(* Logix 5000 project; controller HP_SSC01 vendor 1 type 14 code 67 rev 17.7; software revision 17.01; part 14 of 15 *)
(* tags used below, declared in another part *)
   A_C2_0200 : ALIAS FOR S_C2_FaultSafety.0;
   A_C2_0201 : ALIAS FOR S_C2_FaultSafety.1;
   A_C2_0202 : ALIAS FOR S_C2_FaultSafety.2;
   A_C2_0203 : ALIAS FOR S_C2_FaultSafety.3;
   A_C2_0204 : ALIAS FOR S_C2_FaultSafety.4;
   A_C2_0206 : ALIAS FOR S_C2_FaultSafety.6;
   A_C2_0208 : ALIAS FOR S_C2_FaultSafety.8;
   A_C2_0209 : ALIAS FOR S_C2_FaultSafety.9;
   A_C2_0210 : ALIAS FOR S_C2_FaultSafety.10;
   A_C2_0211 : ALIAS FOR S_C2_FaultSafety.11;
   A_C2_0216 : ALIAS FOR S_C2_FaultSafety.16;
   A_C2_0217 : ALIAS FOR S_C2_FaultSafety.17;
   A_C2_0220 : ALIAS FOR S_C2_FaultSafety.20;
   A_C3_0200 : ALIAS FOR S_C3_FaultSafety.0;
   A_C3_0201 : ALIAS FOR S_C3_FaultSafety.1;
   A_C3_0202 : ALIAS FOR S_C3_FaultSafety.2;
   A_C3_0203 : ALIAS FOR S_C3_FaultSafety.3;
   A_C3_0204 : ALIAS FOR S_C3_FaultSafety.4;
   A_C3_0206 : ALIAS FOR S_C3_FaultSafety.6;
   A_C3_0208 : ALIAS FOR S_C3_FaultSafety.8;
   A_C3_0209 : ALIAS FOR S_C3_FaultSafety.9;
   A_C3_0210 : ALIAS FOR S_C3_FaultSafety.10;
   A_C3_0211 : ALIAS FOR S_C3_FaultSafety.11;
   A_C3_0216 : ALIAS FOR S_C3_FaultSafety.16;
   A_C3_0217 : ALIAS FOR S_C3_FaultSafety.17;
   A_C3_0218 : ALIAS FOR S_C3_FaultSafety.18;
   A_C3_0219 : ALIAS FOR S_C3_FaultSafety.19;
   A_C3_0220 : ALIAS FOR S_C3_FaultSafety.20;
   A_C3_0221 : ALIAS FOR S_C3_FaultSafety.21;
   A_C3_0222 : ALIAS FOR S_C3_FaultSafety.22;
   A_C3_0223 : ALIAS FOR S_C3_FaultSafety.23;
   A_C3_0224 : ALIAS FOR S_C3_FaultSafety.24;
   A_C3_0230 : ALIAS FOR S_C3_FaultSafety.30;
   A_C3_0231 : ALIAS FOR S_C3_FaultSafety.31;
   A_S01_0104 : ALIAS FOR System_FaultSafeIO.4;
   A_S01_0122 : ALIAS FOR System_FaultSafeIO.22;
   C03_SafeMemory : Udt_Carsl_SafeData;
   C2_EvacInPositionTest : DINT;
   Multiplier : DINT;
   none : BOOL;
   RCS_CMD_EvacToStation : BOOL;
   RCS_SafeMemory_S01 : Udt_RCS_SafeData;
   RCS_SyncMotionEnable : BOOL;
   S1_C3_SafeOffFdbkRIN : REDUNDANT_INPUT;
   S_C1_ModeRemote : BOOL;
   S_C2_AtEvacSpeed : BOOL;
   S_C2_BrakeTest : BOOL;
   S_C2_CircuitReset : BOOL;
   S_C2_CircuitReset_Pulse : TIMER;
   S_C2_DrawBridge_LS1 : ALIAS FOR SSC01_Safe2:I.Pt02Data;
   S_C2_DrawBridge_LS2 : ALIAS FOR SSC01_Safe2:I.Pt03Data;
   S_C2_DrawbridgeInputOK : BOOL;
   S_C2_DrawbridgeRIN : REDUNDANT_INPUT;
   S_C2_DumpTest : BOOL;
   S_C2_EvacOK : BOOL;
   S_C2_ExecuteInputOK : BOOL;
   S_C2_ExecutePB : BOOL;
   S_C2_FaultReset : BOOL;
   S_C2_FaultSafety : DINT;
   S_C2_FaultSafety_OK : BOOL;
   S_C2_FaultStandard : DINT;
   S_C2_FaultStandard_OK : BOOL;
   S_C2_FW_LocalOK : BOOL;
   S_C2_InEvacPosition : BOOL;
   S_C2_MaintEnable : BOOL;
   S_C2_MCC2_LIM_MCR : ALIAS FOR C2_Safe:O.Pt04Data;
   S_C2_ModeLocal : BOOL;
   S_C2_ModeRemote : BOOL;
   S_C2_MotionEnabled : BOOL;
   S_C2_MOTN_EXEC_RIN : REDUNDANT_INPUT;
   S_C2_MOTN_EXEC_SS_A : ALIAS FOR C2_Safe:I.Pt02Data;
   S_C2_MOTN_EXEC_SS_B : ALIAS FOR C2_Safe:I.Pt03Data;
   S_C2_MotorActualPositionX1000 : DINT;
   S_C2_MotorAverageVelocityX1000 : DINT;
   S_C2_MStop : EMERGENCY_STOP;
   S_C2_MSTOP_A : ALIAS FOR C2_Safe:I.Pt06Data;
   S_C2_MSTOP_B : ALIAS FOR C2_Safe:I.Pt07Data;
   S_C2_MSTOP_InputOK : BOOL;
   S_C2_MSTOP_LT : ALIAS FOR C2_Safe:O.Pt02Data;
   S_C2_OIT_FaultReset : BOOL;
   S_C2_ONS : DINT;
   S_C2_ONS_CircuitFault : BOOL;
   S_C2_ONS_Status : BOOL;
   S_C2_OutputEnable : BOOL;
   S_C2_PressureOK : ALIAS FOR C2_Safe:I.Pt05Data;
   S_C2_ResetTOF : TIMER;
   S_C2_SAFE_FDBK_Aux1 : BOOL;
   S_C2_SAFE_FDBK_Aux2 : BOOL;
   S_C2_SAFE_OFF_FDBK1 : ALIAS FOR C2_Safe:I.Pt01Data;
   S_C2_SAFE_OFF_FDBK2 : ALIAS FOR C2_Safe:I.Pt00Data;
   S_C2_SafeOff_ROUT : REDUNDANT_OUTPUT;
   S_C2_SafeOffEnabled : BOOL;
   S_C2_SafeOffEngaged : BOOL;
   S_C2_SafeOffFdbkRIN : REDUNDANT_INPUT;
   S_C2_SafeOffInputOK : BOOL;
   S_C2_SAFETY_ENABLE_1 : ALIAS FOR C2_Safe:O.Pt00Data;
   S_C2_SAFETY_ENABLE_2 : ALIAS FOR C2_Safe:O.Pt01Data;
   S_C2_SS_RemoteMode : BOOL;
   S_C2_Stop0_OK : BOOL;
   S_C2_Stop1_OK : BOOL;
   S_C2_Stop1_OK_TOF : TIMER;
   S_C3_AtEvacSpeed : BOOL;
   S_C3_BrakeRelease : ALIAS FOR C3_Safe:O.Pt06Data;
   S_C3_BrakeReleaseSelected : BOOL;
   S_C3_BrakeTest : BOOL;
   S_C3_CircuitReset : BOOL;
   S_C3_CircuitReset_Pulse : TIMER;
   S_C3_DrawBridge_LS1 : ALIAS FOR SSC01_Safe2:I.Pt06Data;
   S_C3_DrawBridge_LS2 : ALIAS FOR SSC01_Safe2:I.Pt07Data;
   S_C3_DrawbridgeInputOK : BOOL;
   S_C3_DrawbridgeRIN : REDUNDANT_INPUT;
   S_C3_DumpValveRelease : ALIAS FOR C3_Safe:O.Pt05Data;
   S_C3_DumpValveReleaseSelected : BOOL;
   S_C3_EncoderBuffer : DINT[4];
   S_C3_EncoderChange : DINT;
   S_C3_EncoderCounter : DINT;
   S_C3_EncoderCounts : DINT;
   S_C3_EncoderDegree : DINT;
   S_C3_EncoderPositionAtHome : DINT;
   S_C3_EncoderPositionAtHomeSet : BOOL;
   S_C3_EncoderRev : DINT;
   S_C3_EncoderRevX1000 : DINT;
   S_C3_EncoderTemp : DINT;
   S_C3_EncoderTemp2 : DINT;
   S_C3_EvacOK : BOOL;
   S_C3_ExecuteInputOK : BOOL;
   S_C3_ExecutePB : BOOL;
   S_C3_FaultReset : BOOL;
   S_C3_FaultSafety : DINT;
   S_C3_FaultSafety_OK : BOOL;
   S_C3_FaultStandard_OK : BOOL;
   S_C3_FaultTimer : TIMER[8];
   S_C3_Homed : BOOL;
   S_C3_HomeInputStatus : BOOL;
   S_C3_HomeSafePE : ALIAS FOR C3_Safe:I.Pt04Data;
   S_C3_InEvacPosition : BOOL;
   S_C3_ModeLocal : BOOL;
   S_C3_ModeRemote : BOOL;
   S_C3_MOTN_EXEC_RIN : REDUNDANT_INPUT;
   S_C3_MOTN_EXEC_SS_A : ALIAS FOR C3_Safe:I.Pt02Data;
   S_C3_MOTN_EXEC_SS_B : ALIAS FOR C3_Safe:I.Pt03Data;
   S_C3_MotorActualPositionX1000 : DINT;
   S_C3_MotorActualPositionX1000MOD60 : DINT;
   S_C3_MotorAverageVelocityX1000 : DINT;
   S_C3_MotorToEncoderError : DINT;
   S_C3_MStop : EMERGENCY_STOP;
   S_C3_MSTOP_A : ALIAS FOR C3_Safe:I.Pt06Data;
   S_C3_MSTOP_B : ALIAS FOR C3_Safe:I.Pt07Data;
   S_C3_MSTOP_InputOK : BOOL;
   S_C3_NearOnPath : BOOL;
   S_C3_NearOnPathHi : DINT;
   S_C3_NearOnPathHiBase : DINT;
   S_C3_NearOnPathLow : DINT;
   S_C3_NearOnPathLowBase : DINT;
   S_C3_OffPath : BOOL;
   S_C3_OnPath : BOOL;
   S_C3_OnPathHi : DINT;
   S_C3_OnPathLow : DINT;
   S_C3_ONS_CircuitFault : BOOL;
   S_C3_ONS_Fault : BOOL;
   S_C3_OutputEnable : BOOL;
   S_C3_PathError : DINT;
   S_C3_PathErrorTest : DINT;
   S_C3_PathErrorTestTemp : DINT;
   S_C3_PathErrorTestTemp2 : DINT;
   S_C3_PathOffset : DINT;
   S_C3_PressureOK : ALIAS FOR C3_Safe:I.Pt05Data;
   S_C3_RemoteBrakeAndHomeSequence : DINT;
   S_C3_ReverseMotionDebounce : TIMER;
   S_C3_SAFE_FDBK_Aux1 : BOOL;
   S_C3_SAFE_FDBK_Aux2 : BOOL;
   S_C3_SAFE_OFF_FDBK1 : ALIAS FOR C3_Safe:I.Pt01Data;
   S_C3_SAFE_OFF_FDBK2 : ALIAS FOR C3_Safe:I.Pt00Data;
   S_C3_SafeOff_ROUT : REDUNDANT_OUTPUT;
   S_C3_SafeOffEnabled : BOOL;
   S_C3_SafeOffEngaged : BOOL;
   S_C3_SafeOffInputOK : BOOL;
   S_C3_SetEncoderHomePosition : BOOL;
   S_C3_WindowAdderTemp1 : DINT;
   S_C3_WindowAdderTemp2 : DINT;
   S_C3_WindowAdderTemp3 : DINT;
   S_EncoderRollover : DINT;
   S_EvacToStationTON : TIMER;
   S_FlashOn : TIMER;
   S_RCS_CMD_FaultReset : BOOL;
   S_RCS_EvacSpeedStart_TON : TIMER;
   S_RCS_MasterPositionDegrees : DINT;
   S_RCS_MotionEnable : BOOL;
   S_System_FaultStandard : DINT;
   SSC_Rail_BypassOK : BOOL;
   SSC_SafeFlt_OK : BOOL;
   SSC_SafetyIO_OK : BOOL;
   SSC_StdFlt_OK : BOOL;
   SSC_Stop0_OK : BOOL;
   SSC_Stop1_OK : BOOL;
(* SafeCarousel2, continued *)

ROUTINE SC230_SafetyInputs   (* ladder *)
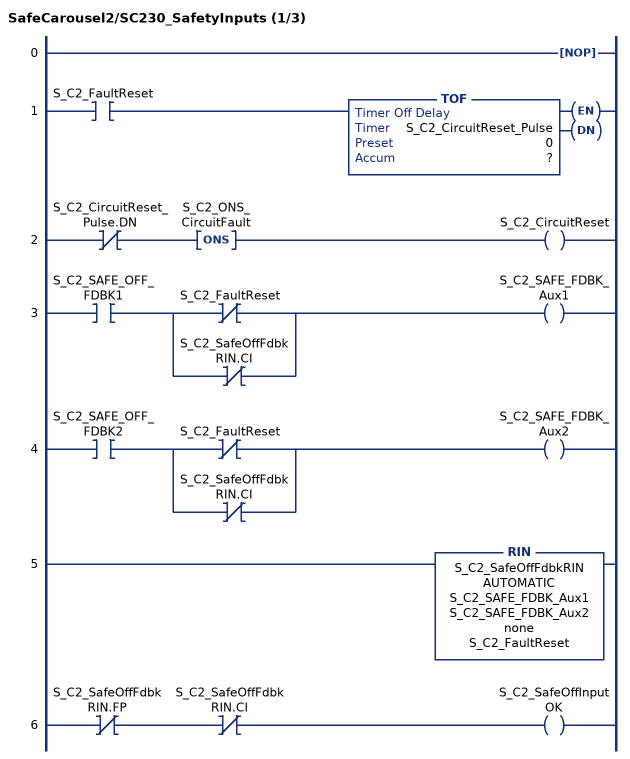
   0: NOP();
   1: XIC(S_C2_FaultReset)TOF(S_C2_CircuitReset_Pulse,?,?);
   2: XIO(S_C2_CircuitReset_Pulse.DN)ONS(S_C2_ONS_CircuitFault)OTE(S_C2_CircuitReset);
   3: XIC(S_C2_SAFE_OFF_FDBK1)[XIO(S_C2_FaultReset) ,XIO(S_C2_SafeOffFdbkRIN.CI) ]OTE(S_C2_SAFE_FDBK_Aux1);
   4: XIC(S_C2_SAFE_OFF_FDBK2)[XIO(S_C2_FaultReset) ,XIO(S_C2_SafeOffFdbkRIN.CI) ]OTE(S_C2_SAFE_FDBK_Aux2);
   5: RIN(S_C2_SafeOffFdbkRIN,AUTOMATIC,S_C2_SAFE_FDBK_Aux1,S_C2_SAFE_FDBK_Aux2,none,S_C2_FaultReset);
   6: XIO(S_C2_SafeOffFdbkRIN.FP)XIO(S_C2_SafeOffFdbkRIN.CI)OTE(S_C2_SafeOffInputOK);
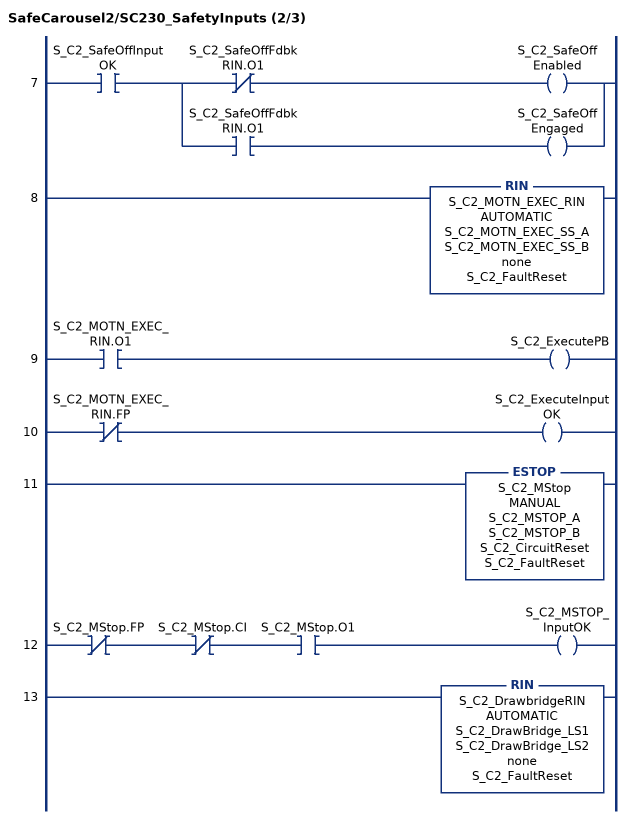
   7: XIC(S_C2_SafeOffInputOK)[XIO(S_C2_SafeOffFdbkRIN.O1) OTE(S_C2_SafeOffEnabled) ,XIC(S_C2_SafeOffFdbkRIN.O1) OTE(S_C2_SafeOffEngaged) ];
   8: RIN(S_C2_MOTN_EXEC_RIN,AUTOMATIC,S_C2_MOTN_EXEC_SS_A,S_C2_MOTN_EXEC_SS_B,none,S_C2_FaultReset);
   9: XIC(S_C2_MOTN_EXEC_RIN.O1)OTE(S_C2_ExecutePB);
   10: XIO(S_C2_MOTN_EXEC_RIN.FP)OTE(S_C2_ExecuteInputOK);
   11: ESTOP(S_C2_MStop,MANUAL,S_C2_MSTOP_A,S_C2_MSTOP_B,S_C2_CircuitReset,S_C2_FaultReset);
   12: XIO(S_C2_MStop.FP)XIO(S_C2_MStop.CI)XIC(S_C2_MStop.O1)OTE(S_C2_MSTOP_InputOK);
   13: RIN(S_C2_DrawbridgeRIN,AUTOMATIC,S_C2_DrawBridge_LS1,S_C2_DrawBridge_LS2,none,S_C2_FaultReset);
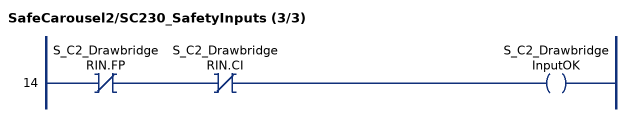
   14: XIO(S_C2_DrawbridgeRIN.FP)XIO(S_C2_DrawbridgeRIN.CI)OTE(S_C2_DrawbridgeInputOK);
END_ROUTINE

ROUTINE SC235_SafetyOutputs   (* ladder *)
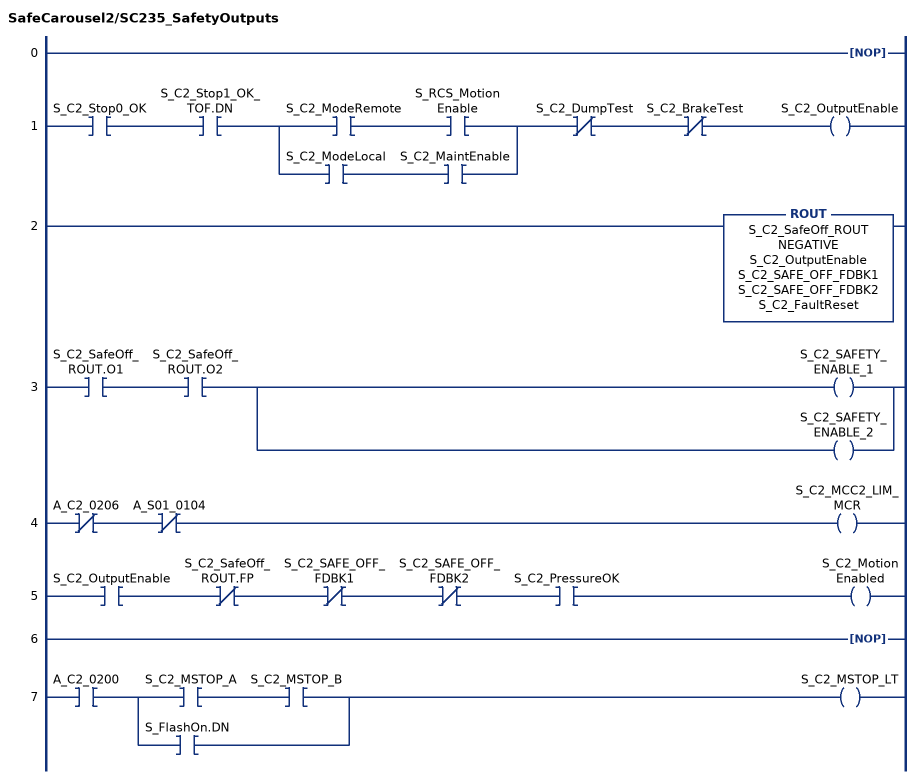
   0: NOP();
   1: XIC(S_C2_Stop0_OK)XIC(S_C2_Stop1_OK_TOF.DN)[XIC(S_C2_ModeRemote) XIC(S_RCS_MotionEnable) ,XIC(S_C2_ModeLocal) XIC(S_C2_MaintEnable) ]XIO(S_C2_DumpTest)XIO(S_C2_BrakeTest)OTE(S_C2_OutputEnable);
   2: ROUT(S_C2_SafeOff_ROUT,NEGATIVE,S_C2_OutputEnable,S_C2_SAFE_OFF_FDBK1,S_C2_SAFE_OFF_FDBK2,S_C2_FaultReset);
   3: XIC(S_C2_SafeOff_ROUT.O1)XIC(S_C2_SafeOff_ROUT.O2)[OTE(S_C2_SAFETY_ENABLE_1) ,OTE(S_C2_SAFETY_ENABLE_2) ];
   4: XIO(A_C2_0206)XIO(A_S01_0104)OTE(S_C2_MCC2_LIM_MCR);
   5: XIC(S_C2_OutputEnable)XIO(S_C2_SafeOff_ROUT.FP)XIO(S_C2_SAFE_OFF_FDBK1)XIO(S_C2_SAFE_OFF_FDBK2)XIC(S_C2_PressureOK)OTE(S_C2_MotionEnabled);
   6: NOP();
   7: XIC(A_C2_0200)[XIC(S_C2_MSTOP_A) XIC(S_C2_MSTOP_B) ,XIC(S_FlashOn.DN) ]OTE(S_C2_MSTOP_LT);
END_ROUTINE

ROUTINE SC240_Status   (* ladder *)
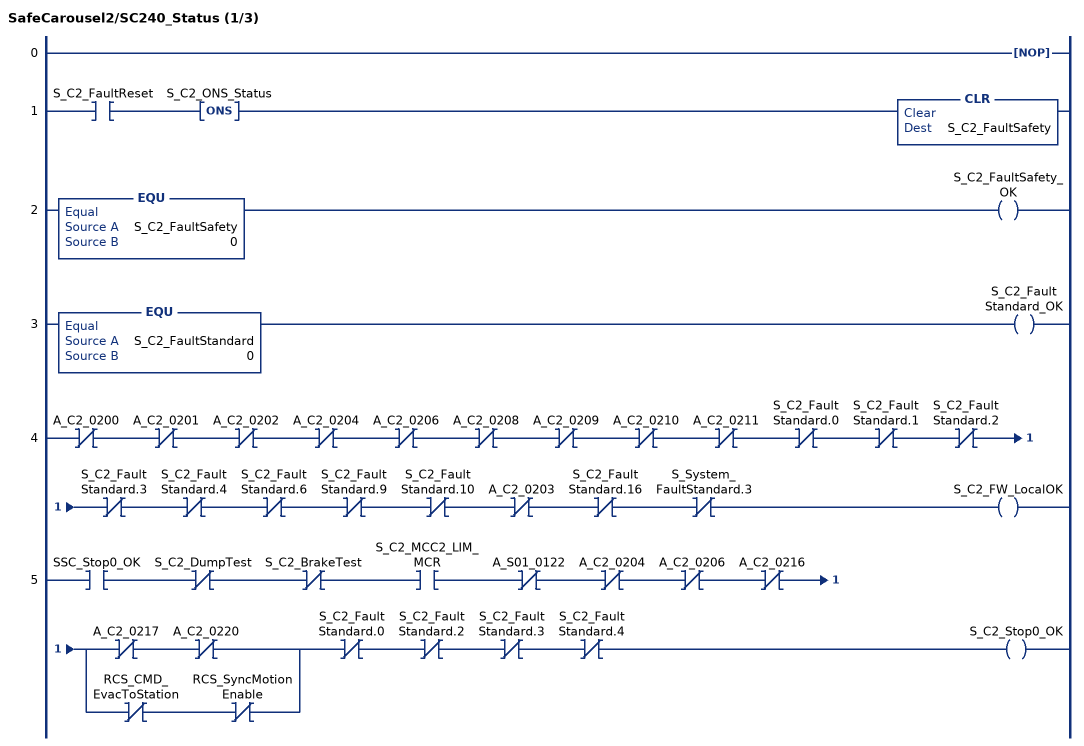
   0: NOP();
   1: XIC(S_C2_FaultReset)ONS(S_C2_ONS_Status)CLR(S_C2_FaultSafety);
   2: EQU(S_C2_FaultSafety,0)OTE(S_C2_FaultSafety_OK);
   3: EQU(S_C2_FaultStandard,0)OTE(S_C2_FaultStandard_OK);
   4: XIO(A_C2_0200)XIO(A_C2_0201)XIO(A_C2_0202)XIO(A_C2_0204)XIO(A_C2_0206)XIO(A_C2_0208)XIO(A_C2_0209)XIO(A_C2_0210)XIO(A_C2_0211)XIO(S_C2_FaultStandard.0)XIO(S_C2_FaultStandard.1)XIO(S_C2_FaultStandard.2)XIO(S_C2_FaultStandard.3)XIO(S_C2_FaultStandard.4)XIO(S_C2_FaultStandard.6)XIO(S_C2_FaultStandard.9)XIO(S_C2_FaultStandard.10)XIO(A_C2_0203)XIO(S_C2_FaultStandard.16)XIO(S_System_FaultStandard.3)OTE(S_C2_FW_LocalOK);
   5: XIC(SSC_Stop0_OK)XIO(S_C2_DumpTest)XIO(S_C2_BrakeTest)XIC(S_C2_MCC2_LIM_MCR)XIO(A_S01_0122)XIO(A_C2_0204)XIO(A_C2_0206)XIO(A_C2_0216)[XIO(A_C2_0217) XIO(A_C2_0220) ,XIO(RCS_CMD_EvacToStation) XIO(RCS_SyncMotionEnable) ]XIO(S_C2_FaultStandard.0)XIO(S_C2_FaultStandard.2)XIO(S_C2_FaultStandard.3)XIO(S_C2_FaultStandard.4)OTE(S_C2_Stop0_OK);
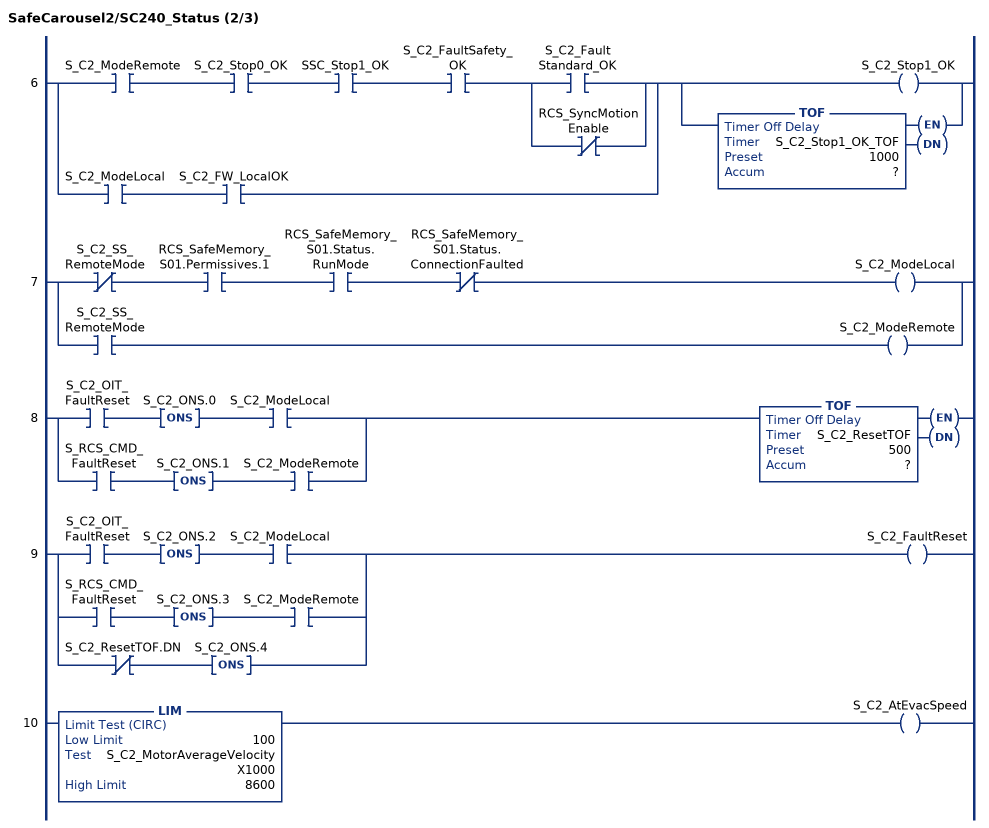
   6: [XIC(S_C2_ModeRemote) XIC(S_C2_Stop0_OK) XIC(SSC_Stop1_OK) XIC(S_C2_FaultSafety_OK) [XIC(S_C2_FaultStandard_OK) ,XIO(RCS_SyncMotionEnable) ] ,XIC(S_C2_ModeLocal) XIC(S_C2_FW_LocalOK) ][OTE(S_C2_Stop1_OK) ,TOF(S_C2_Stop1_OK_TOF,?,?) ];
   7: [XIO(S_C2_SS_RemoteMode) XIC(RCS_SafeMemory_S01.Permissives.1) XIC(RCS_SafeMemory_S01.Status.RunMode) XIO(RCS_SafeMemory_S01.Status.ConnectionFaulted) OTE(S_C2_ModeLocal) ,XIC(S_C2_SS_RemoteMode) OTE(S_C2_ModeRemote) ];
   8: [XIC(S_C2_OIT_FaultReset) ONS(S_C2_ONS.0) XIC(S_C2_ModeLocal) ,XIC(S_RCS_CMD_FaultReset) ONS(S_C2_ONS.1) XIC(S_C2_ModeRemote) ]TOF(S_C2_ResetTOF,?,?);
   9: [XIC(S_C2_OIT_FaultReset) ONS(S_C2_ONS.2) XIC(S_C2_ModeLocal) ,XIC(S_RCS_CMD_FaultReset) ONS(S_C2_ONS.3) XIC(S_C2_ModeRemote) ,XIO(S_C2_ResetTOF.DN) ONS(S_C2_ONS.4) ]OTE(S_C2_FaultReset);
   10: LIM(100,S_C2_MotorAverageVelocityX1000,8600)OTE(S_C2_AtEvacSpeed);
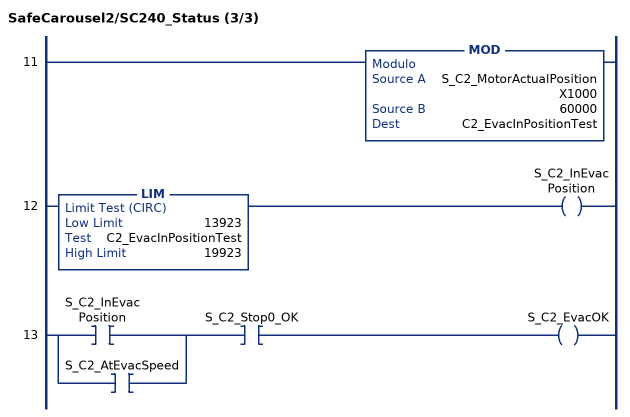
   11: MOD(S_C2_MotorActualPositionX1000,60000,C2_EvacInPositionTest);
   12: LIM(13923,C2_EvacInPositionTest,19923)OTE(S_C2_InEvacPosition);
   13: [XIC(S_C2_InEvacPosition) ,XIC(S_C2_AtEvacSpeed) ]XIC(S_C2_Stop0_OK)OTE(S_C2_EvacOK);
END_ROUTINE
END_PROGRAM

PROGRAM SafeCarousel3   (* main routine SC300_Main *)

ROUTINE SC300_Main   (* ladder *)
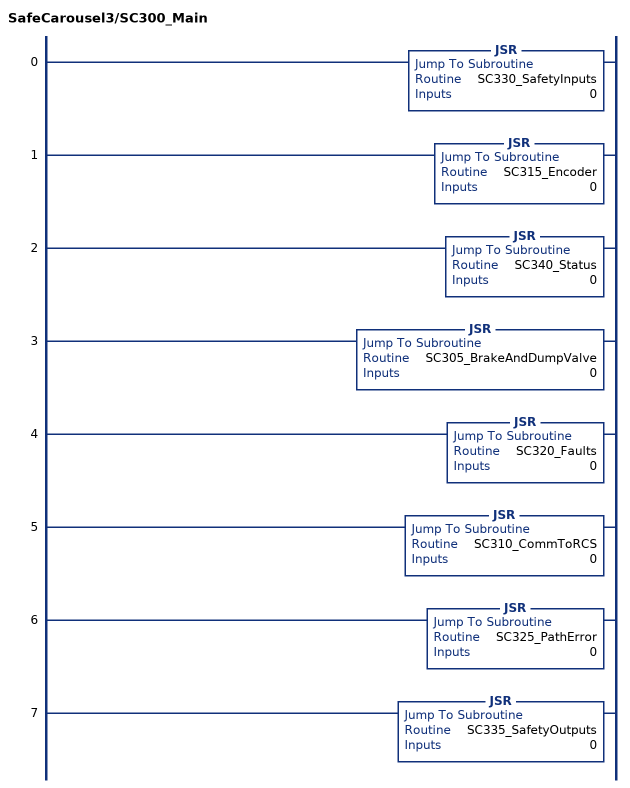
   0: JSR(SC330_SafetyInputs,0);
   1: JSR(SC315_Encoder,0);
   2: JSR(SC340_Status,0);
   3: JSR(SC305_BrakeAndDumpValve,0);
   4: JSR(SC320_Faults,0);
   5: JSR(SC310_CommToRCS,0);
   6: JSR(SC325_PathError,0);
   7: JSR(SC335_SafetyOutputs,0);
END_ROUTINE

ROUTINE SC305_BrakeAndDumpValve   (* ladder *)
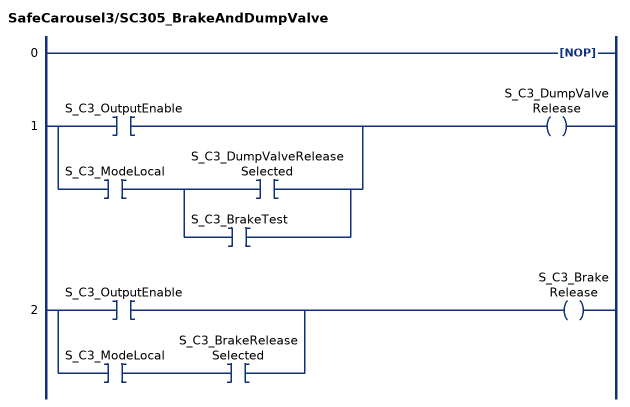
   0: NOP();
   1: [XIC(S_C3_OutputEnable) ,XIC(S_C3_ModeLocal) [XIC(S_C3_DumpValveReleaseSelected) ,XIC(S_C3_BrakeTest) ] ]OTE(S_C3_DumpValveRelease);
   2: [XIC(S_C3_OutputEnable) ,XIC(S_C3_ModeLocal) XIC(S_C3_BrakeReleaseSelected) ]OTE(S_C3_BrakeRelease);
END_ROUTINE

ROUTINE SC310_CommToRCS   (* ladder *)
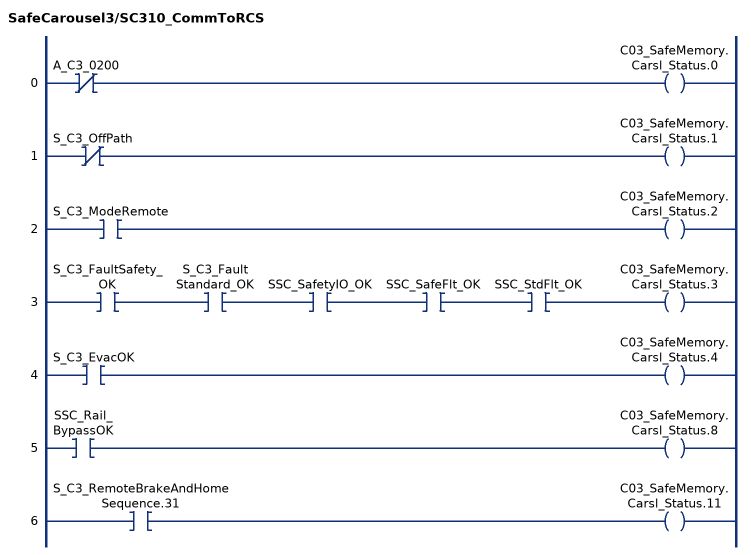
   0: XIO(A_C3_0200)OTE(C03_SafeMemory.Carsl_Status.0);
   1: XIO(S_C3_OffPath)OTE(C03_SafeMemory.Carsl_Status.1);
   2: XIC(S_C3_ModeRemote)OTE(C03_SafeMemory.Carsl_Status.2);
   3: XIC(S_C3_FaultSafety_OK)XIC(S_C3_FaultStandard_OK)XIC(SSC_SafetyIO_OK)XIC(SSC_SafeFlt_OK)XIC(SSC_StdFlt_OK)OTE(C03_SafeMemory.Carsl_Status.3);
   4: XIC(S_C3_EvacOK)OTE(C03_SafeMemory.Carsl_Status.4);
   5: XIC(SSC_Rail_BypassOK)OTE(C03_SafeMemory.Carsl_Status.8);
   6: XIC(S_C3_RemoteBrakeAndHomeSequence.31)OTE(C03_SafeMemory.Carsl_Status.11);
END_ROUTINE

ROUTINE SC315_Encoder   (* ladder *)
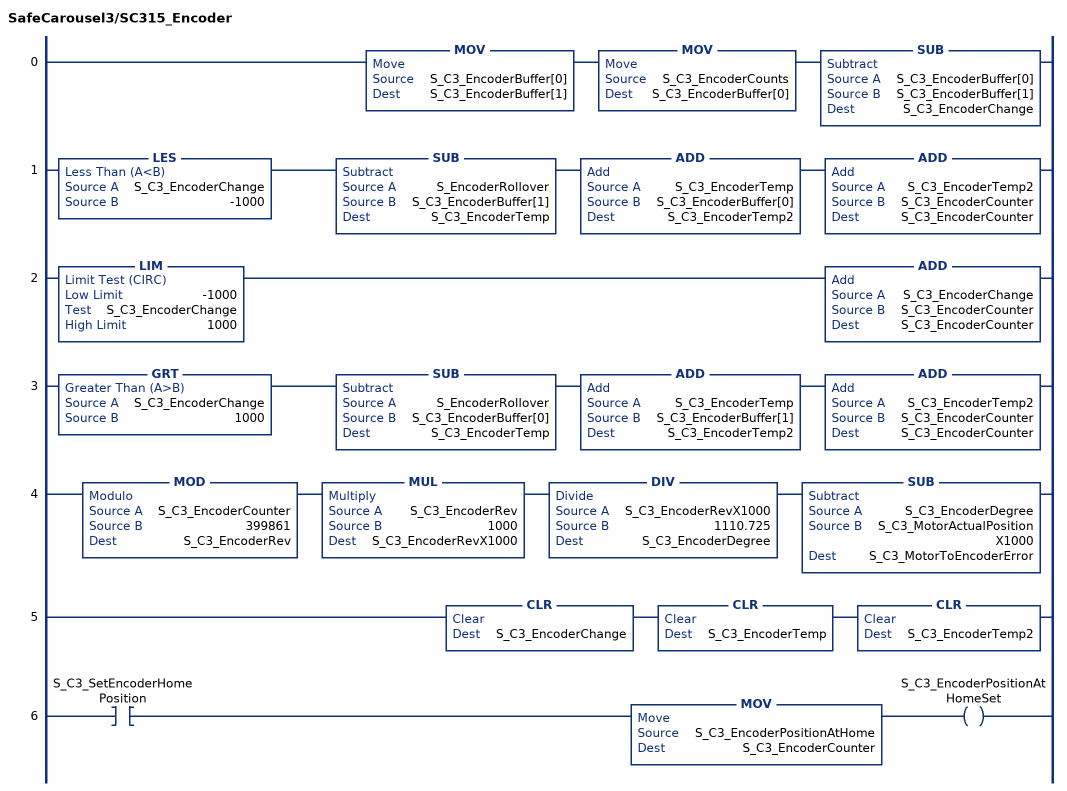
   0: MOV(S_C3_EncoderBuffer[0],S_C3_EncoderBuffer[1])MOV(S_C3_EncoderCounts,S_C3_EncoderBuffer[0])SUB(S_C3_EncoderBuffer[0],S_C3_EncoderBuffer[1],S_C3_EncoderChange);
   1: LES(S_C3_EncoderChange,-1000)SUB(S_EncoderRollover,S_C3_EncoderBuffer[1],S_C3_EncoderTemp)ADD(S_C3_EncoderTemp,S_C3_EncoderBuffer[0],S_C3_EncoderTemp2)ADD(S_C3_EncoderTemp2,S_C3_EncoderCounter,S_C3_EncoderCounter);
   2: LIM(-1000,S_C3_EncoderChange,1000)ADD(S_C3_EncoderChange,S_C3_EncoderCounter,S_C3_EncoderCounter);
   3: GRT(S_C3_EncoderChange,1000)SUB(S_EncoderRollover,S_C3_EncoderBuffer[0],S_C3_EncoderTemp)ADD(S_C3_EncoderTemp,S_C3_EncoderBuffer[1],S_C3_EncoderTemp2)ADD(S_C3_EncoderTemp2,S_C3_EncoderCounter,S_C3_EncoderCounter);
   4: MOD(S_C3_EncoderCounter,399861,S_C3_EncoderRev)MUL(S_C3_EncoderRev,1000,S_C3_EncoderRevX1000)DIV(S_C3_EncoderRevX1000,1110.725,S_C3_EncoderDegree)SUB(S_C3_EncoderDegree,S_C3_MotorActualPositionX1000,S_C3_MotorToEncoderError);
   5: CLR(S_C3_EncoderChange)CLR(S_C3_EncoderTemp)CLR(S_C3_EncoderTemp2);
   6: XIC(S_C3_SetEncoderHomePosition)MOV(S_C3_EncoderPositionAtHome,S_C3_EncoderCounter)OTE(S_C3_EncoderPositionAtHomeSet);
END_ROUTINE

ROUTINE SC320_Faults   (* ladder *)
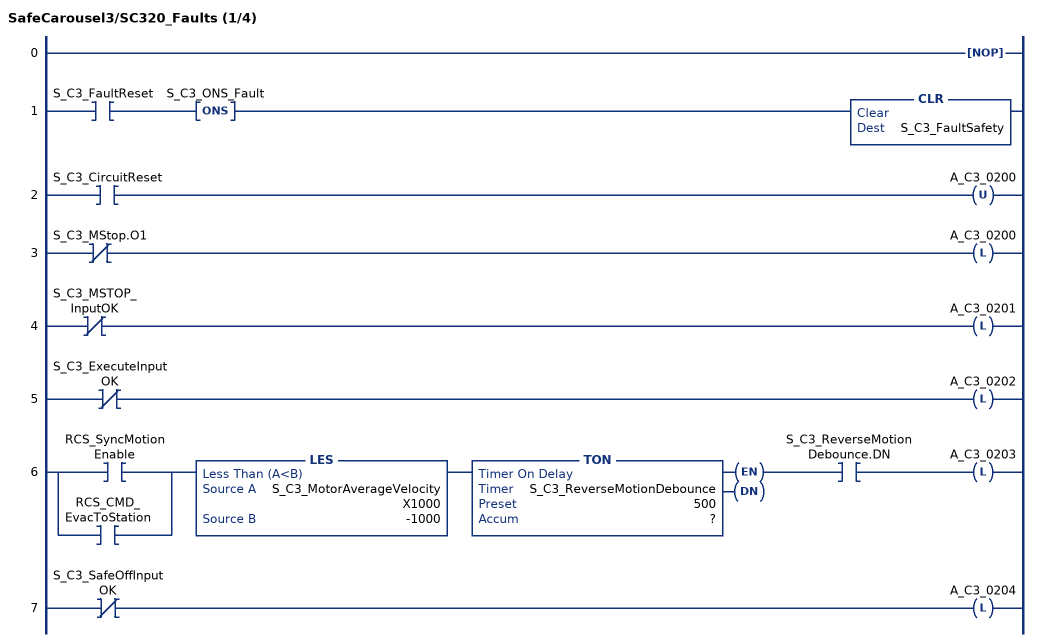
   0: NOP();
   1: XIC(S_C3_FaultReset)ONS(S_C3_ONS_Fault)CLR(S_C3_FaultSafety);
   2: XIC(S_C3_CircuitReset)OTU(A_C3_0200);
   3: XIO(S_C3_MStop.O1)OTL(A_C3_0200);
   4: XIO(S_C3_MSTOP_InputOK)OTL(A_C3_0201);
   5: XIO(S_C3_ExecuteInputOK)OTL(A_C3_0202);
   6: [XIC(RCS_SyncMotionEnable) ,XIC(RCS_CMD_EvacToStation) ]LES(S_C3_MotorAverageVelocityX1000,-1000)TON(S_C3_ReverseMotionDebounce,?,?)XIC(S_C3_ReverseMotionDebounce.DN)OTL(A_C3_0203);
   7: XIO(S_C3_SafeOffInputOK)OTL(A_C3_0204);
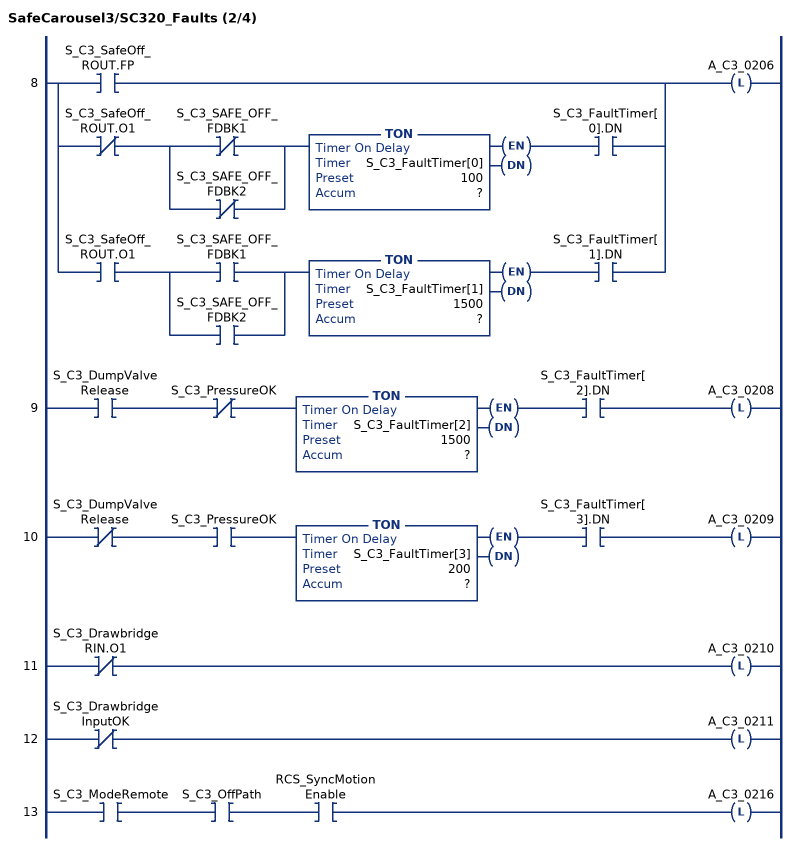
   8: [XIC(S_C3_SafeOff_ROUT.FP) ,XIO(S_C3_SafeOff_ROUT.O1) [XIO(S_C3_SAFE_OFF_FDBK1) ,XIO(S_C3_SAFE_OFF_FDBK2) ] TON(S_C3_FaultTimer[0],?,?) XIC(S_C3_FaultTimer[0].DN) ,XIC(S_C3_SafeOff_ROUT.O1) [XIC(S_C3_SAFE_OFF_FDBK1) ,XIC(S_C3_SAFE_OFF_FDBK2) ] TON(S_C3_FaultTimer[1],?,?) XIC(S_C3_FaultTimer[1].DN) ]OTL(A_C3_0206);
   9: XIC(S_C3_DumpValveRelease)XIO(S_C3_PressureOK)TON(S_C3_FaultTimer[2],?,?)XIC(S_C3_FaultTimer[2].DN)OTL(A_C3_0208);
   10: XIO(S_C3_DumpValveRelease)XIC(S_C3_PressureOK)TON(S_C3_FaultTimer[3],?,?)XIC(S_C3_FaultTimer[3].DN)OTL(A_C3_0209);
   11: XIO(S_C3_DrawbridgeRIN.O1)OTL(A_C3_0210);
   12: XIO(S_C3_DrawbridgeInputOK)OTL(A_C3_0211);
   13: XIC(S_C3_ModeRemote)XIC(S_C3_OffPath)XIC(RCS_SyncMotionEnable)OTL(A_C3_0216);
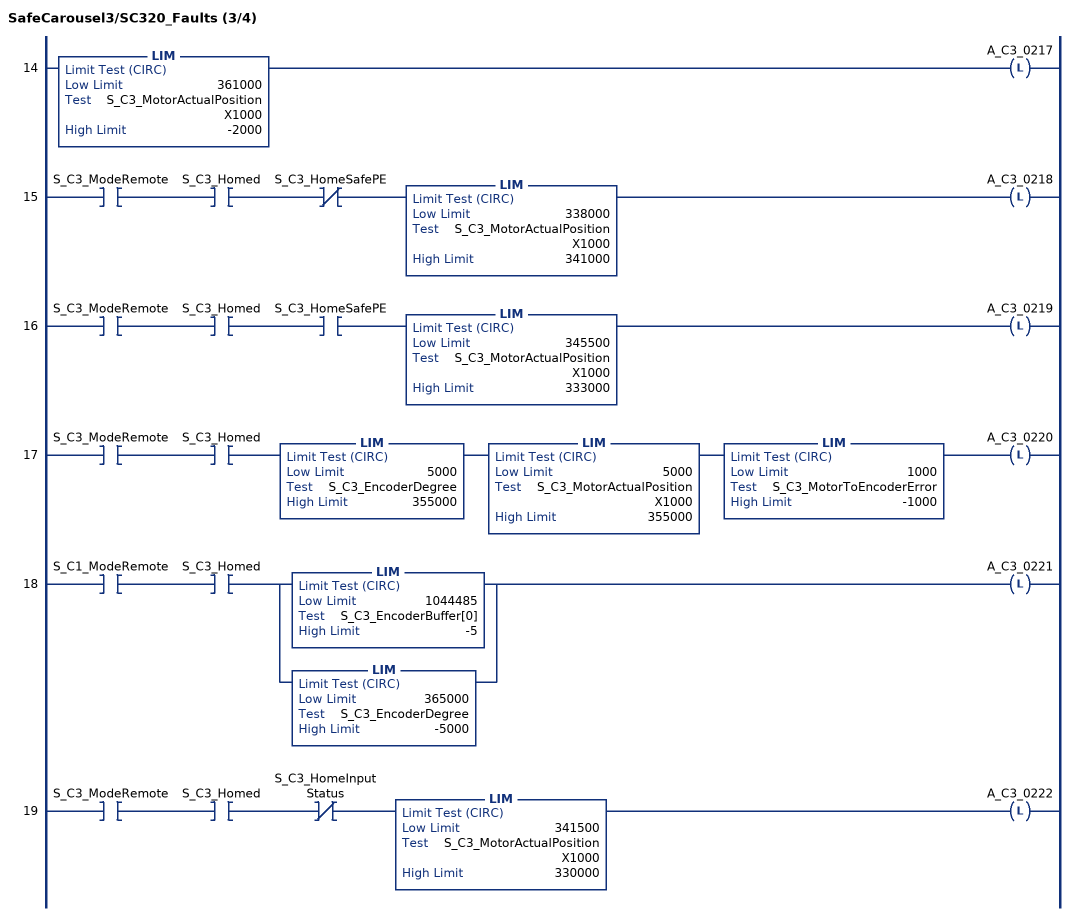
   14: LIM(361000,S_C3_MotorActualPositionX1000,-2000)OTL(A_C3_0217);
   15: XIC(S_C3_ModeRemote)XIC(S_C3_Homed)XIO(S_C3_HomeSafePE)LIM(338000,S_C3_MotorActualPositionX1000,341000)OTL(A_C3_0218);
   16: XIC(S_C3_ModeRemote)XIC(S_C3_Homed)XIC(S_C3_HomeSafePE)LIM(345500,S_C3_MotorActualPositionX1000,333000)OTL(A_C3_0219);
   17: XIC(S_C3_ModeRemote)XIC(S_C3_Homed)LIM(5000,S_C3_EncoderDegree,355000)LIM(5000,S_C3_MotorActualPositionX1000,355000)LIM(1000,S_C3_MotorToEncoderError,-1000)OTL(A_C3_0220);
   18: XIC(S_C1_ModeRemote)XIC(S_C3_Homed)[LIM(1044485,S_C3_EncoderBuffer[0],-5) ,LIM(365000,S_C3_EncoderDegree,-5000) ]OTL(A_C3_0221);
   19: XIC(S_C3_ModeRemote)XIC(S_C3_Homed)XIO(S_C3_HomeInputStatus)LIM(341500,S_C3_MotorActualPositionX1000,330000)OTL(A_C3_0222);
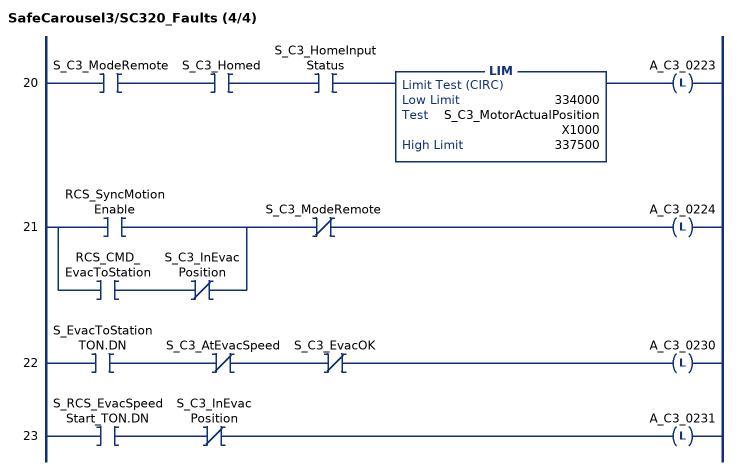
   20: XIC(S_C3_ModeRemote)XIC(S_C3_Homed)XIC(S_C3_HomeInputStatus)LIM(334000,S_C3_MotorActualPositionX1000,337500)OTL(A_C3_0223);
   21: [XIC(RCS_SyncMotionEnable) ,XIC(RCS_CMD_EvacToStation) XIO(S_C3_InEvacPosition) ]XIO(S_C3_ModeRemote)OTL(A_C3_0224);
   22: XIC(S_EvacToStationTON.DN)XIO(S_C3_AtEvacSpeed)XIO(S_C3_EvacOK)OTL(A_C3_0230);
   23: XIC(S_RCS_EvacSpeedStart_TON.DN)XIO(S_C3_InEvacPosition)OTL(A_C3_0231);
END_ROUTINE

ROUTINE SC325_PathError   (* ladder *)
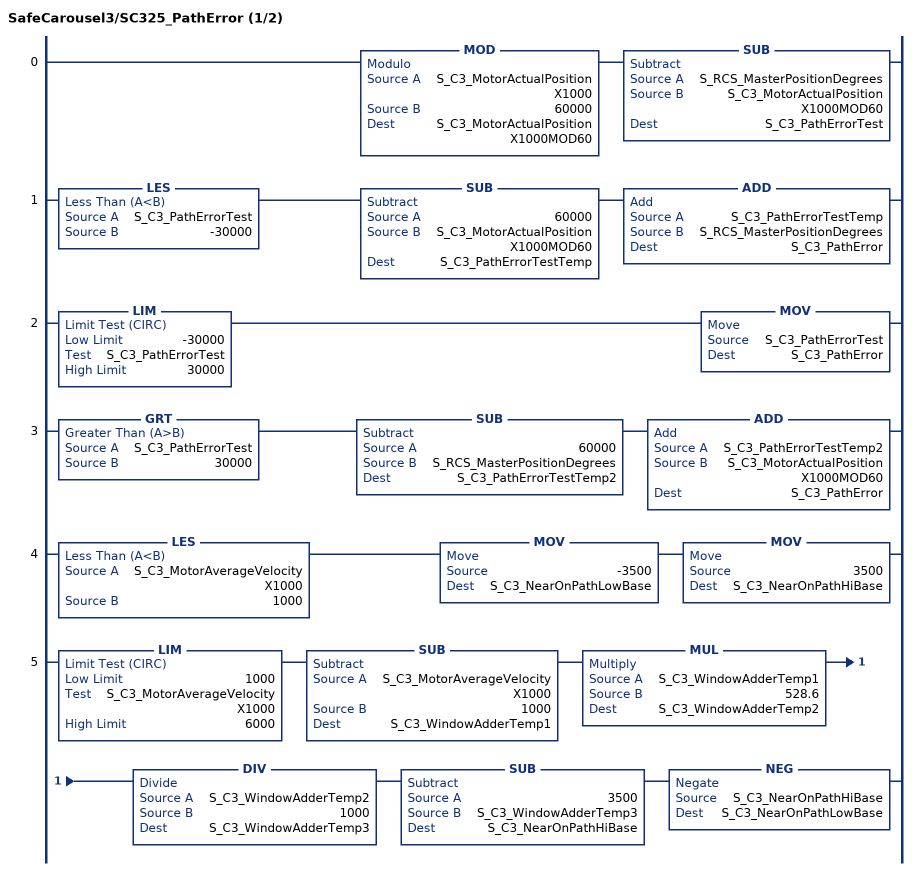
   0: MOD(S_C3_MotorActualPositionX1000,60000,S_C3_MotorActualPositionX1000MOD60)SUB(S_RCS_MasterPositionDegrees,S_C3_MotorActualPositionX1000MOD60,S_C3_PathErrorTest);
   1: LES(S_C3_PathErrorTest,-30000)SUB(60000,S_C3_MotorActualPositionX1000MOD60,S_C3_PathErrorTestTemp)ADD(S_C3_PathErrorTestTemp,S_RCS_MasterPositionDegrees,S_C3_PathError);
   2: LIM(-30000,S_C3_PathErrorTest,30000)MOV(S_C3_PathErrorTest,S_C3_PathError);
   3: GRT(S_C3_PathErrorTest,30000)SUB(60000,S_RCS_MasterPositionDegrees,S_C3_PathErrorTestTemp2)ADD(S_C3_PathErrorTestTemp2,S_C3_MotorActualPositionX1000MOD60,S_C3_PathError);
   4: LES(S_C3_MotorAverageVelocityX1000,1000)MOV(-3500,S_C3_NearOnPathLowBase)MOV(3500,S_C3_NearOnPathHiBase);
   5: LIM(1000,S_C3_MotorAverageVelocityX1000,6000)SUB(S_C3_MotorAverageVelocityX1000,1000,S_C3_WindowAdderTemp1)MUL(S_C3_WindowAdderTemp1,528.6,S_C3_WindowAdderTemp2)DIV(S_C3_WindowAdderTemp2,1000,S_C3_WindowAdderTemp3)SUB(3500,S_C3_WindowAdderTemp3,S_C3_NearOnPathHiBase)NEG(S_C3_NearOnPathHiBase,S_C3_NearOnPathLowBase);
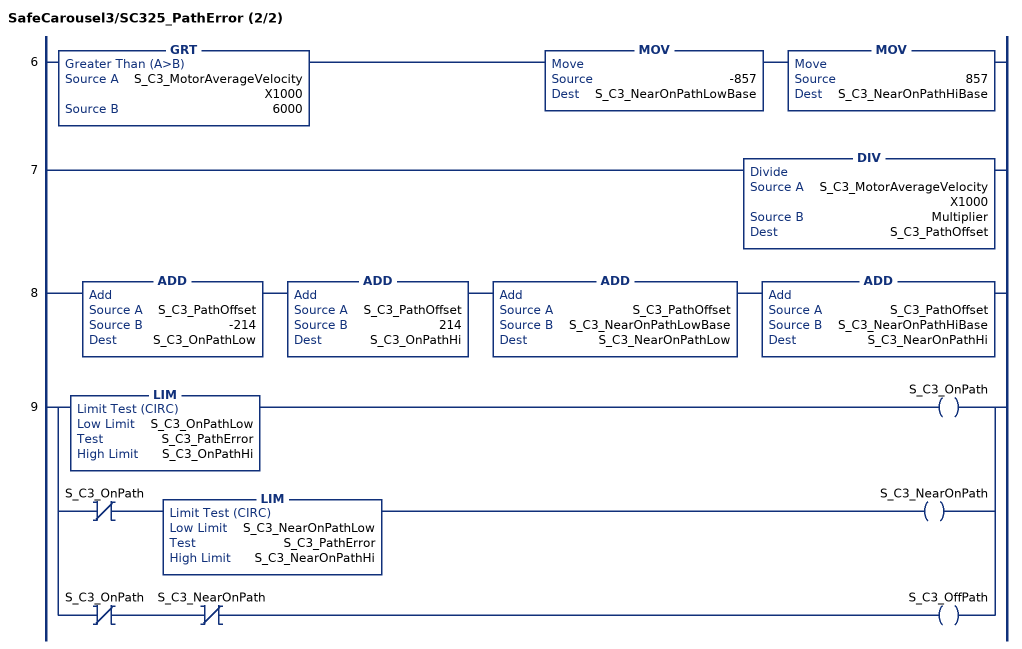
   6: GRT(S_C3_MotorAverageVelocityX1000,6000)MOV(-857,S_C3_NearOnPathLowBase)MOV(857,S_C3_NearOnPathHiBase);
   7: DIV(S_C3_MotorAverageVelocityX1000,Multiplier,S_C3_PathOffset);
   8: ADD(S_C3_PathOffset,-214,S_C3_OnPathLow)ADD(S_C3_PathOffset,214,S_C3_OnPathHi)ADD(S_C3_PathOffset,S_C3_NearOnPathLowBase,S_C3_NearOnPathLow)ADD(S_C3_PathOffset,S_C3_NearOnPathHiBase,S_C3_NearOnPathHi);
   9: [LIM(S_C3_OnPathLow,S_C3_PathError,S_C3_OnPathHi) OTE(S_C3_OnPath) ,XIO(S_C3_OnPath) LIM(S_C3_NearOnPathLow,S_C3_PathError,S_C3_NearOnPathHi) OTE(S_C3_NearOnPath) ,XIO(S_C3_OnPath) XIO(S_C3_NearOnPath) OTE(S_C3_OffPath) ];
END_ROUTINE

ROUTINE SC330_SafetyInputs   (* ladder *)
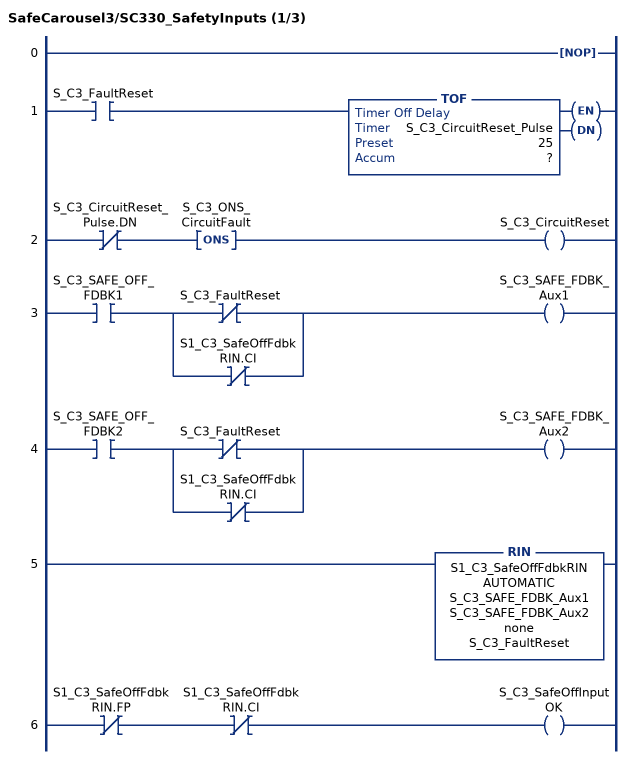
   0: NOP();
   1: XIC(S_C3_FaultReset)TOF(S_C3_CircuitReset_Pulse,?,?);
   2: XIO(S_C3_CircuitReset_Pulse.DN)ONS(S_C3_ONS_CircuitFault)OTE(S_C3_CircuitReset);
   3: XIC(S_C3_SAFE_OFF_FDBK1)[XIO(S_C3_FaultReset) ,XIO(S1_C3_SafeOffFdbkRIN.CI) ]OTE(S_C3_SAFE_FDBK_Aux1);
   4: XIC(S_C3_SAFE_OFF_FDBK2)[XIO(S_C3_FaultReset) ,XIO(S1_C3_SafeOffFdbkRIN.CI) ]OTE(S_C3_SAFE_FDBK_Aux2);
   5: RIN(S1_C3_SafeOffFdbkRIN,AUTOMATIC,S_C3_SAFE_FDBK_Aux1,S_C3_SAFE_FDBK_Aux2,none,S_C3_FaultReset);
   6: XIO(S1_C3_SafeOffFdbkRIN.FP)XIO(S1_C3_SafeOffFdbkRIN.CI)OTE(S_C3_SafeOffInputOK);
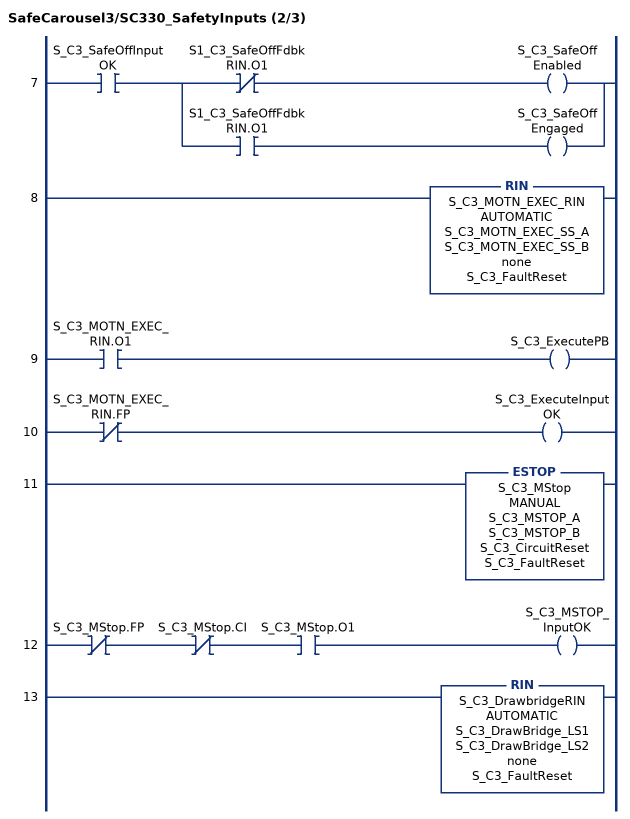
   7: XIC(S_C3_SafeOffInputOK)[XIO(S1_C3_SafeOffFdbkRIN.O1) OTE(S_C3_SafeOffEnabled) ,XIC(S1_C3_SafeOffFdbkRIN.O1) OTE(S_C3_SafeOffEngaged) ];
   8: RIN(S_C3_MOTN_EXEC_RIN,AUTOMATIC,S_C3_MOTN_EXEC_SS_A,S_C3_MOTN_EXEC_SS_B,none,S_C3_FaultReset);
   9: XIC(S_C3_MOTN_EXEC_RIN.O1)OTE(S_C3_ExecutePB);
   10: XIO(S_C3_MOTN_EXEC_RIN.FP)OTE(S_C3_ExecuteInputOK);
   11: ESTOP(S_C3_MStop,MANUAL,S_C3_MSTOP_A,S_C3_MSTOP_B,S_C3_CircuitReset,S_C3_FaultReset);
   12: XIO(S_C3_MStop.FP)XIO(S_C3_MStop.CI)XIC(S_C3_MStop.O1)OTE(S_C3_MSTOP_InputOK);
   13: RIN(S_C3_DrawbridgeRIN,AUTOMATIC,S_C3_DrawBridge_LS1,S_C3_DrawBridge_LS2,none,S_C3_FaultReset);
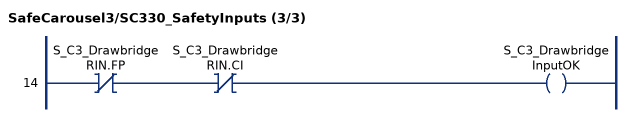
   14: XIO(S_C3_DrawbridgeRIN.FP)XIO(S_C3_DrawbridgeRIN.CI)OTE(S_C3_DrawbridgeInputOK);
END_ROUTINE
